{attribute 'qualified_only'}

TYPE e_SafetyState :
(
	Reset := 100,
	Session:=101,
	Connection:=102,
	Parameter:=103,
	Data:=104,
	Shutdown:=105,
	ShutDownDeactivate:=106
);
END_TYPE

(* stored: Version 1.1.0.1, ProductVersion 3.1.4024.12
   DUT e_SafetyState: Id {203baff3-5dc8-470a-86c7-d7eb94858424} *)
